Universal Robots PolyScope program: debounce_force.urp

Program debounce_force (installation=default directory=/home/ur/ursim-current/programs/idealMFG/debounce createdIn=5.16.0 lastSavedIn=5.17.2 robotSerialNumber=20236899999)
Calibrated DH parameters: a=[0, -0.862, -0.7287, 0, 0, 0]; d=[0.2363, 0, 0, 0.201, 0.1593, 0.1543]; alpha=[1.570796, 0, 0, 1.570796, -1.570796, 0]; deltaTheta=[0, 0, 0, 0, 0, 0]
InitVariablesNode
Robot Program (runOnlyOnce=false)
  Folder numbers to initialize
    'put this in the before start sequence'
    fx_thresh := 20
    fy_thresh := 15
    fz_thresh := 10
    f_count_thresh := 10
    fx_count := 0
    fy_count := 0
    fz_count := 0
    fx_contact := False
    fy_contact := False
    fz_contact := False
  Folder measurement 
    'force measuring and contact detection thread, put this in a thread'
    raw_force := get_tcp_force()
    f_x := raw_force[0]
    f_y := raw_force[1]
    f_z := raw_force[2]
    Folder x
      If norm(f_x)≥fx_thresh
        fx_count := fx_count+1
      Else 
        fx_count := 0
      If fx_count≥f_count_thresh
        fx_contact := True
      Else 
        fx_contact := False
    Folder y
      If norm(f_y)≥fy_thresh
        fy_count := fy_count+1
      Else 
        fy_count := 0
      If fy_count≥f_count_thresh
        fy_contact := True
      Else 
        fy_contact := False
    Folder z
      If norm(f_z)≥fz_thresh
        fz_count := fz_count+1
      Else 
        fz_count := 0
      If fz_count≥f_count_thresh
        fz_contact := True
      Else 
        fz_contact := False
    Script: sync()
